(* PLC project Generated.project, CODESYS CODESYS V3.5 SP19 Patch 1 *)
(* stored: creationDateTime 2026-08-26T00:48:09.010815, modificationDateTime 2026-08-26T00:48:09.010815 *)

(* values of E_WinchFinalInterlockState: DISABLED: Desactive / Hors service; READY: Pret / Etat nominal; WAIT_BRAKE_COMMAND_CONFIRMATION: Attente confirmation feedback frein; WAIT_STEP_DELAY: Temporisation changement de palier; WAIT_RESTART_DELAY: Temporisation anti-court-cycle redemarrage; FAULT: Etat de defaut *)

{attribute 'qualified_only'}
{attribute 'strict'}
TYPE E_WinchFinalInterlockState : (DISABLED := 0, READY := 1, WAIT_BRAKE_COMMAND_CONFIRMATION := 2, WAIT_STEP_DELAY := 3, WAIT_RESTART_DELAY := 4, FAULT := 5);
END_TYPE
